FUNCTION_BLOCK ControlPanel (* Composite Function Block Type *)
  (* Standard: 61499-2 *)
  (* Version 0.0, 2/16/2019, Sandeep Patil, nxtControl GmbH, template *)
  PACKAGE Main;
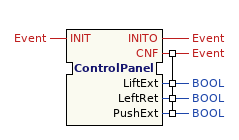
  EVENT_INPUT
    INIT; (* Initialization Request *)
  END_EVENT
  EVENT_OUTPUT
    INITO; (* Initialization Confirm *)
    CNF WITH PushExt, LeftRet, LiftExt; (* Execution Confirmation *)
  END_EVENT
  VAR_OUTPUT
    LiftExt : BOOL;
    LeftRet : BOOL;
    PushExt : BOOL;
  END_VAR
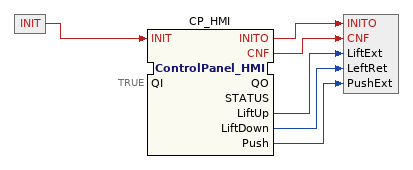
  FBS
    CP_HMI : ControlPanel_HMI(QI := TRUE);
  END_FBS
  EVENT_CONNECTIONS
    INIT TO CP_HMI.INIT;
    CP_HMI.INITO TO INITO;
    CP_HMI.CNF TO CNF;
  END_CONNECTIONS
  DATA_CONNECTIONS
    CP_HMI.LiftUp TO LiftExt;
    CP_HMI.LiftDown TO LeftRet;
    CP_HMI.Push TO PushExt;
  END_CONNECTIONS
END_FUNCTION_BLOCK
